// TIA Portal V16 export
// export: Created 2021-09-08T12:46:08.7452919Z, ExportSetting WithDefaults, DisplayName Totally Integrated Automation Portal, DisplayVersion V16 Update 3, DisplayName TIA Portal Version Control Interface, DisplayVersion V16 Update 2, DisplayName TIA Portal Openness, DisplayVersion V16 Update 3, DisplayName TIA Portal Teamcenter Gateway, DisplayVersion V16, DisplayName STEP 7 Professional, DisplayVersion V16 Update 3, DisplayName STEP 7 Safety, DisplayVersion V16, DisplayName WinCC Advanced, DisplayVersion V16 Update 3
FUNCTION_BLOCK "TON_200ms"   // FB9, FBD
{ S7_Optimized_Access := 'TRUE' }
VERSION : 0.1
// stored: AutoNumber true, IsIECCheckEnabled false, IsRetainMemResEnabled false, MemoryReserve 100, SetENOAutomatically false, UDAEnableTagReadback false
   VAR_INPUT
      In : Bool;
      PT : Time;
   END_VAR
   VAR_OUTPUT
      ET : Time;
      Q : Bool;
   END_VAR
BEGIN

REGION Network 1: Увеличение текущего времени
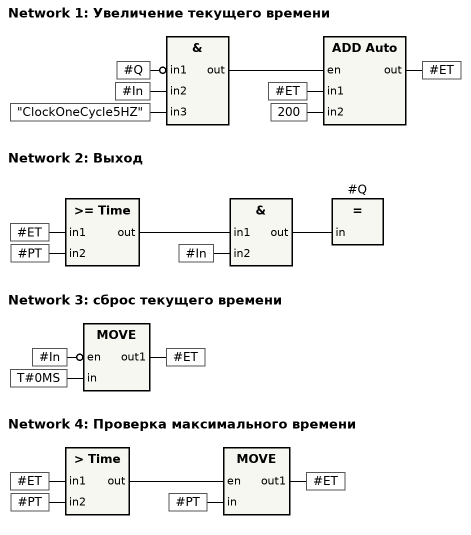
   IF NOT #Q AND #In AND "ClockOneCycle5HZ" THEN #ET := #ET + 200; END_IF;
END_REGION

REGION Network 2: Выход
   #Q := (#ET >= #PT) AND #In;
END_REGION

REGION Network 3: сброс текущего времени
   IF NOT #In THEN #ET := T#0MS; END_IF;
END_REGION

REGION Network 4: Проверка максимального времени
   IF #ET > #PT THEN #ET := #PT; END_IF;
END_REGION
END_FUNCTION_BLOCK
